(* CoDeSys 2.3 export: CHECKDIVDWORD.EXP *)

(* POU CheckDivDWord, ST *)
FUNCTION CheckDivDWord : DWORD
VAR_INPUT
	divisor: DWORD;
END_VAR
VAR
END_VAR
(* @TEXT_IMPLEMENTATION := 'ST' *)
IF divisor = 0 THEN
	CheckDivDWord := 1;
ELSE
	CheckDivDWord := divisor;
END_IF
END_FUNCTION
